FUNCTION F_Derotatorposition : LREAL
VAR_INPUT
	// azimuth in degrees
	azimuth:		LREAL;
	// latitude in degrees
	latitude: 		LREAL;
	// declination in degrees
	declination:	LREAL;
	// elevation in degrees
	elevation:		LREAL;
END_VAR
VAR
	parallactic_angle:	LREAL;
	az, lat, delta, pa:	LREAL;
END_VAR
VAR CONSTANT
	d2r:	LREAL := PI/180.0;
	r2d:	LREAL := 180.0/PI;
END_VAR

(*
calculation for the derotator position
source: GRE-KIS-MAN-0008 GREGOR: Derotator Manual
returns derotatorposition in degrees
*)
// convert azimuth to radians
az := azimuth * d2r;
// convert latitude to radians
lat := latitude * d2r;
// convert declination to radians
delta := declination * d2r;

// calculate the parallactic angle

IF ABS(COS(delta)) < 1E-3 THEN
	pa := 0.0;
ELSE
	pa := ASIN(SIN(az) * COS(lat) / COS(delta));
END_IF

// convert parallactic angle to degrees
parallactic_angle := pa * r2d;

F_Derotatorposition := parallactic_angle + azimuth + elevation;

END_FUNCTION

(* stored: Version 1.1.0.1, ProductVersion 3.1.4024.9
   POU F_Derotatorposition: Id {60bb6b84-d38a-49fc-a26b-76a4adc375c0}, SpecialFunc None *)
